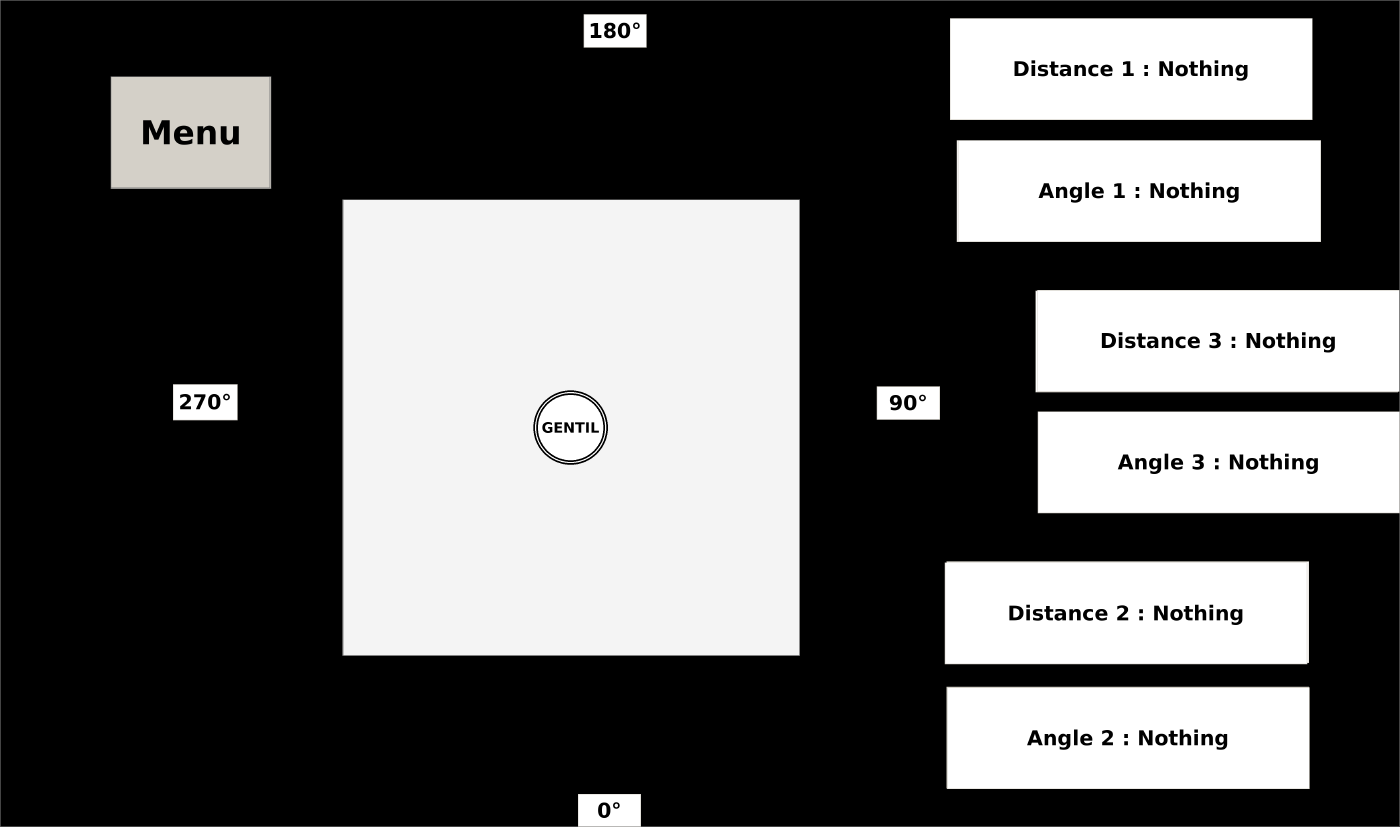
VISUALIZATION V_Balise  // 2454x1451
    Line (1000,750) (1000,50)
    Line (1000,750) (1700,750)
    Line (1000,750) (300,750)
    Line (1000,750) (1000,1450)
    Textfield (1665,32 635x178), "Distance1 : %10.1f", text variable: G_Balise.lrDistance_1, invisible if: ITInterruption.balise.Nothing1
    Textfield (1677,246 635x178), "Angle1 : %10.1f", text variable: G_Balise.lrAngle_1, invisible if: ITInterruption.balise.Nothing1
    Textfield (1659,1205 635x178), "Angle 2 : %10.1f", text variable: G_Balise.lrAngle_2, invisible if: ITInterruption.balise.Nothing2
    Textfield (1659,985 635x178), "Distance2 : %10.1f", text variable: G_Balise.lrDistance_2, invisible if: ITInterruption.balise.Nothing2
    Textfield (1537,678 110x58), "90°", colour toggle: ITInterruption.balise.Angle90deg
    Textfield (1023,25 110x58), "180°", colour toggle: ITInterruption.balise.Angle180deg
    Textfield (303,674 113x63), "270°", colour toggle: ITInterruption.balise.Angle270deg
    Textfield (1013,1393 110x58), "0°", colour toggle: ITInterruption.balise.Angle0deg
    Textfield (1656,987 635x178), "Distance 2 : Nothing", text variable: G_Balise.lrDistance_2, invisible if: not ITInterruption.balise.Nothing2
    Textfield (1665,32 635x178), "Distance 1 : Nothing", text variable: G_Balise.lrDistance_1, invisible if: not ITInterruption.balise.Nothing1
    Pie (600,350 800x800), invisible if: ITInterruption.balise.Angle0deg
    Pie (600,350 800x800), invisible if: ITInterruption.balise.Angle90deg
    Pie (602,350 800x800), invisible if: ITInterruption.balise.Angle180deg
    Pie (601,350 800x800), invisible if: ITInterruption.balise.Angle270deg
    Ellipse (935,685 130x130), "Méchant", invisible if: ITInterruption.balise.Nothing2
        p3528305787: ITInterruption.balise.posiX2
        p2773130477: ITInterruption.balise.posiY2
        p874137650: ITInterruption.balise.posiX2
        p1126004900: ITInterruption.balise.posiY2
    Ellipse (935,685 130x130), "Méchant", invisible if: ITInterruption.balise.Nothing1
        p3528305787: ITInterruption.balise.posiX1
        p2773130477: ITInterruption.balise.posiY1
        p874137650: ITInterruption.balise.posiX1
        p1126004900: ITInterruption.balise.posiY1
    Line (1000,750) (1000,750), colour toggle: ITInterruption.balise.D1_40cm, invisible if: ITInterruption.balise.Nothing1
        p874137650: ITInterruption.balise.posiX1
        p1126004900: ITInterruption.balise.posiY1
    Line (1000,750) (1000,750), colour toggle: ITInterruption.balise.D2_40cm, invisible if: ITInterruption.balise.Nothing2
        p874137650: ITInterruption.balise.posiX2
        p1126004900: ITInterruption.balise.posiY2
    Textfield (1815,510 635x178), "Distance3 : %10.1f", text variable: G_Balise.ArrayEnnemi [2,1], invisible if: ITInterruption.balise.Nothing3
    Textfield (1819,722 635x178), "Angle 3 : %10.1f", text variable: G_Balise.lrAngle_2, invisible if: ITInterruption.balise.Nothing3
    Textfield (1818,509 635x178), "Distance 3 : Nothing", text variable: G_Balise.lrDistance_3, invisible if: not ITInterruption.balise.Nothing3
    Ellipse (935,685 130x130), "Méchant", invisible if: ITInterruption.balise.Nothing3
        p3528305787: ITInterruption.balise.posiX3
        p2773130477: ITInterruption.balise.posiY3
        p874137650: ITInterruption.balise.posiX3
        p1126004900: ITInterruption.balise.posiY3
    Line (1000,750) (1000,750), colour toggle: ITInterruption.balise.D3_40cm, invisible if: ITInterruption.balise.Nothing3
        p874137650: ITInterruption.balise.posiX3
        p1126004900: ITInterruption.balise.posiY3
    Ellipse (940,690 120x120), "GENTIL"
    Textfield (1819,722 635x178), "Angle 3 : Nothing", text variable: G_Balise.lrAngle_3, invisible if: not ITInterruption.balise.Nothing3
    Textfield (1680,246 635x178), "Angle 1 : Nothing", text variable: G_Balise.lrAngle_1, invisible if: not ITInterruption.balise.Nothing1
    Textfield (1660,1206 635x178), "Angle 2 : Nothing", text variable: G_Balise.lrAngle_2, invisible if: not ITInterruption.balise.Nothing2
    Button (194,134 281x197), "Menu"
        OnMouseDown: change screen: V_Menu
END_VISUALIZATION

(* stored: Version 1.1.0.1, ProductVersion 3.1.4024.12
   Visu V_Balise: Id {21c1c8fe-ee69-411e-b597-24c78f248dd4} *)
